(* PLC project Library, CODESYS V3.5 *)
(* stored: creationDateTime 2022-10-04T11:36:41 *)
(* capital C, and genuinely in the schema *)

FUNCTION_BLOCK P
  VAR_INPUT
    In : Axis;
  END_VAR

;
END_FUNCTION_BLOCK
